// TIA Portal V18 export
// export: Created 2025-12-01T12:38:06.0721095Z, ExportSetting None, DisplayName Totally Integrated Automation Portal, DisplayVersion V18 Update 5, DisplayName TIA Portal Openness, DisplayVersion V18 Update 5, DisplayName TIA Portal Teamcenter Gateway, DisplayVersion V18, DisplayName TIA Portal Version Control Interface, DisplayVersion V18, DisplayName STEP 7 Professional, DisplayVersion V18 Update 5, DisplayName STEP 7 Safety, DisplayVersion V18, DisplayName WinCC Professional, DisplayVersion V18 Update 5
DATA_BLOCK "ST10_SysInput"   // DB1001
{ S7_Optimized_Access := 'TRUE' }
// stored: AutoNumber false, MemoryReserve 100
   VAR
      HMI_Button : Struct
         ControlOn : Bool := false;   // HMI_上电按钮
         ControlOff : Bool;   // HMI_断电按钮
         MachineStart : Bool := false;   // HMI_设备启动按钮
         MachineStop : Bool := false;   // HMI_设备停止按钮
         ResetButton : Bool := false;   // HMI_复位按钮
         "Manual/Auto" : Bool := false;   // HMI_手/自动切换按钮
         SafetyGateUnlock : Bool := false;   // HMI_安全门解锁按钮
         "E-Stop" : Bool := false;   // HMI_急停
      END_STRUCT;
      Sys : Struct
         iCircuitBreakerOK1 : Bool;   // 电子断路器 OK
         iCircuitBreakerOK2 : Bool;
         iPressure : Bool;   // 气压监控
      END_STRUCT;
      "iE-StopPB" : Array[1..20] of Bool;   // 急停按钮PB
      iSafetyGatFeedBack : Array[1..20] of Bool;   // 安全门
      iSafetydoorLockingFeedBack : Array[1..20] of Bool;   // 安全门反馈
      iMaterieldoorLockingFeedBack : Array[1..20] of Bool;   // 安全门反馈
   END_VAR
BEGIN
END_DATA_BLOCK
